PROGRAM Stn052_36_Stn123MainMergePrestop
VAR
	//correct
	{attribute 'TcLinkToOSO' := '.iPuckPresent    :=  <0,1,2>TIIB[N27S00 (AL1332)]^N27S01 (AL2341)^TxPDO^input byte 1;
								 .iBufferFull   :=  <0,1,2>TIIB[N27S00 (AL1332)]^N27S01 (AL2341)^TxPDO^input byte 3;
								 .oStopLower    :=  <0,1,1>TIIB[N27S00 (AL1332)]^N27S05 (EX260)^RxPDO^output byte 1'}	
	fbConvStop: FB_ConvStop;
END_VAR

//  This code instantiates a component that is implimented as a common function block
//    Note that I/O is linked directly to I/O variables inside the named instance

gStn052_36_Stn123MainMergePrestop.ConvRunning := gConsumed_SafetyInterfaceConv.MtrRunning.Enc054Mtr05;

fbConvStop(
	pStn := ADR(gStn052),
	pCmp := ADR(gStn052_36_Stn123MainMergePrestop),
	pUpstreamStop := 0,
	pStateTraceBuffer := ADR(gStn052_StateTraceBuffer),
	pStateTraceFifo := ADR(gStn052_StateTraceFifo),
	pStats := ADR(gStn052_02_Stats));

END_PROGRAM

(* stored: Version 1.1.0.1, ProductVersion 3.1.4024.6
   POU Stn052_36_Stn123MainMergePrestop: Id {26bc5b8a-230d-4ffc-9bcf-60a1264f93e7}, SpecialFunc None *)
